// TIA Portal V20 export
DATA_BLOCK "TEST"   // DB501
// stored: Access Published, MemoryReserve 100, Namespace Unit1
   VAR
      Test : Array[0..100] of Bool;
      TestRange : Array[0..100] of LReal;
      jangBit : Bool;
      KSGbit : Bool;
   END_VAR
BEGIN
   TestRange[0] := 1.0;
END_DATA_BLOCK
